{attribute 'linkalways'} 
{attribute 'no_explicit_call' := 'This FB is a CLASS and must be accessed using methods or properties'}
{attribute 'enable_dynamic_creation'}
FUNCTION_BLOCK GraphFrameworkApi IMPLEMENTS I_RpcApi, I_HostGraphs, I_EventEmitter
VAR
	graphFramework : I_GraphFramework;
	eventEmitter : EventEmitter;
	graphHost : GraphHost(THIS^, eventEmitter);
	createGraphRpcHandler : CreateGraphRpcHandler;
	createGraphMultiUserRpcHandler : CreateGraphMultiUserRpcHandler;
	getStatusRpcHandler : GetStatusRpcHandler;
	getBlueprintsRpcHandler : GetBlueprintsRpcHandler;
	getContentValueHandler : GetContentValueHandler;
	updateParameterValueHandler : UpdateParameterValueHandler;
END_VAR

METHOD PUBLIC CyclicCall
VAR_INPUT
END_VAR
graphHost.Execute();
END_METHOD

METHOD FB_exit : BOOL
VAR_INPUT
	bInCopyCode : BOOL; // if TRUE, the exit method is called for exiting an instance that is copied afterwards (online change).
END_VAR
IF bInCopyCode THEN
	RETURN;
END_IF

graphs.DisposeAll();
END_METHOD

METHOD FB_init : BOOL
VAR_INPUT
	bInitRetains : BOOL; // if TRUE, the retain variables are initialized (warm start / cold start)
	bInCopyCode : BOOL;  // if TRUE, the instance afterwards gets moved into the copy code (online change)
	GraphFramework : I_GraphFramework;
END_VAR
THIS^.graphFramework := GraphFramework;

getBlueprintsRpcHandler.Initialize(GraphFramework.NodeFactory);
getStatusRpcHandler.Initialize(graphHost);
createGraphRpcHandler.Initialize(GraphFramework, graphHost);
createGraphMultiUserRpcHandler.Initialize(GraphFramework, graphHost);
getContentValueHandler.Initialize(graphHost);
updateParameterValueHandler.Initialize(graphHost);
END_METHOD

PROPERTY PUBLIC Graphs : I_Graphs
GET
Graphs := graphHost;
END_GET
END_PROPERTY

METHOD PUBLIC OffEvent
VAR_INPUT
	EventName : T_MaxString;
	EventHandler : I_EventHandler;
END_VAR
eventEmitter.OffEvent(EventName, EventHandler);
END_METHOD

METHOD PUBLIC OnceEvent
VAR_INPUT
	EventName : T_MaxString;
	EventHandler : I_EventHandler;
END_VAR
eventEmitter.OnceEvent(EventName, EventHandler);
END_METHOD

METHOD PUBLIC OnEvent
VAR_INPUT
	EventName : T_MaxString;
	EventHandler : I_EventHandler;
END_VAR
eventEmitter.OnEvent(EventName, EventHandler);
END_METHOD

METHOD RegisterAsynchronousRpcHandlersWith
VAR_INPUT
	Host : I_HostAsynchronousRpcHandlers;
END_VAR
Host.RegisterHandler('CreateGraph', createGraphRpcHandler);
Host.RegisterHandler('CreateGraphMultiUser', createGraphMultiUserRpcHandler);
Host.RegisterHandler('GetStatus', getStatusRpcHandler);
Host.RegisterHandler('GetBlueprints', getBlueprintsRpcHandler);
Host.RegisterHandler('GetContentValue', getContentValueHandler);
Host.RegisterHandler('UpdateParameterValue', updateParameterValueHandler);
END_METHOD

METHOD RegisterSynchronousRpcHandlersWith
VAR_INPUT
	Host : I_HostSynchronousRpcHandlers;
END_VAR
// no implementation
END_METHOD

END_FUNCTION_BLOCK

(* stored: Version 1.1.0.1, ProductVersion 3.1.4024.13
   POU GraphFrameworkApi: Id {bbeaa71e-faa8-4020-94ac-c51b0ba5f637}, SpecialFunc None
   Folder Constructor: Id {3247a7d8-0cdf-41a7-b3ec-00d25e5860b9}
   Folder Destructor: Id {983f8a90-ec8c-4c25-8a21-35742fc4254f}
   Method CyclicCall: Id {61535b54-c31a-0f24-2b44-201dd4ecdbfb}
   Method FB_exit: Id {4eb785ac-97f2-4e9f-bd85-4c70f39c8c99}
   Method FB_init: Id {b497c453-9953-44d6-988c-3152593a8346}
   Property Graphs: Id {7459a2e4-4645-45ec-bd04-a073ccef6af0}
   Get Get: Id {ca3f37f6-bbbb-4cbf-ade0-2bc41c362246}
   Method OffEvent: Id {453e0cb5-5eec-4608-8791-b408daa4f546}
   Method OnceEvent: Id {635c4793-06f8-4101-842b-634a7c40f36e}
   Method OnEvent: Id {8449549f-e645-46b8-856f-f2a55623aa58}
   Method RegisterAsynchronousRpcHandlersWith: Id {16f43e44-1c8f-40af-91d9-0c94f14c9a34}
   Method RegisterSynchronousRpcHandlersWith: Id {9cdb3985-6a52-0982-12b5-714e24122e9a} *)
